(* PLC project Programme MGS_2-07_refactorJOY.project, CODESYS CODESYS V3.5 SP19 Patch 1 *)
(* stored: creationDateTime 2026-06-29T23:37:40.9816606, modificationDateTime 2026-06-29T22:49:33.424 *)

PROGRAM PRG_JOY1
  VAR
    FB_Joystick_0 : FB_Joystick;
  END_VAR

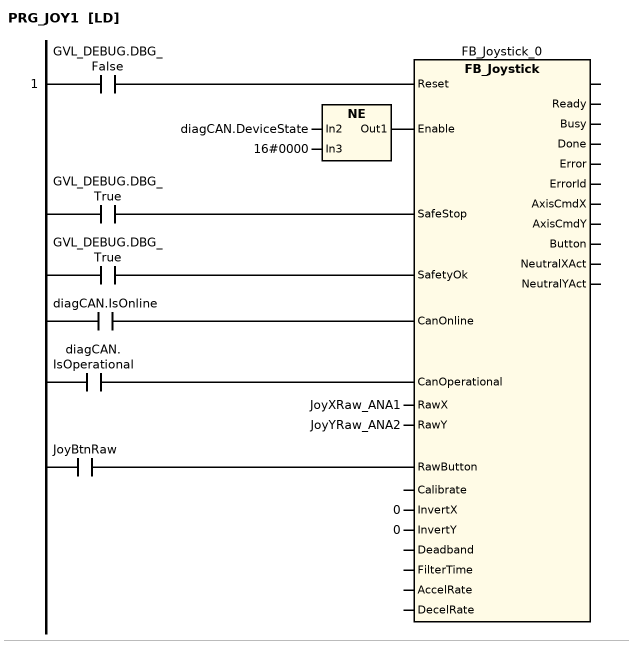
(* LD diagram, written out as Structured Text *)

FB_Joystick_0(Enable := diagCAN.DeviceState <> 16#0000, Reset := GVL_DEBUG.DBG_False, SafeStop := GVL_DEBUG.DBG_True, SafetyOk := GVL_DEBUG.DBG_True, CanOnline := diagCAN.IsOnline, CanOperational := diagCAN.IsOperational, RawX := JoyXRaw_ANA1, RawY := JoyYRaw_ANA2, RawButton := JoyBtnRaw, Calibrate := , InvertX := 0, InvertY := 0, Deadband := , FilterTime := , AccelRate := , DecelRate := );
END_PROGRAM
